// TIA Portal V21 export
VAR_GLOBAL   // PLC tag table "PARTIDAS (ETA)"
   "ETA-P01_FALHA" AT %M60.2 : Bool;
END_VAR
